PROGRAM MAIN
VAR
	nCounter: INT;
END_VAR

nCounter := nCounter + 1;

END_PROGRAM

(* stored: Version 1.1.0.1, ProductVersion 3.1.4024.12
   POU MAIN: Id {602d1ec6-dc89-4712-b3c2-a9222724f330}, SpecialFunc None *)
